// TIA Portal V16 export
// export: Created 2023-01-04T15:44:06.905709Z, ExportSetting WithDefaults, DisplayName Totally Integrated Automation Portal, DisplayVersion V16, DisplayName TIA Portal Version Control Interface, DisplayVersion V16, DisplayName TIA Portal Openness, DisplayVersion V16, DisplayName STEP 7 Professional, DisplayVersion V16, DisplayName STEP 7 Safety, DisplayVersion V16, DisplayName WinCC Advanced, DisplayVersion V16
FUNCTION "Filling_Logik" : Void   // FC5, LAD
{ S7_Optimized_Access := 'TRUE' }
VERSION : 0.1
// stored: AutoNumber true, IsIECCheckEnabled false, SetENOAutomatically false, UDAEnableTagReadback false
   VAR_INPUT
      PS2_Filling_Station : Bool;
      FIC_B102 : Int;
      Liquid_AorB_in_Bottle_ml : Real;
      Liquid_AorB_pct : Int;
      Wait_to_fill : Time;
   END_VAR
   VAR_OUTPUT
      Flow_ml_per_sec : Real;
      FillingData_LiqAorB_ml : Real;
   END_VAR
   VAR_IN_OUT
      Outlet_of_tanks : Bool;
   END_VAR
   VAR_TEMP
      PTRIG1 : Bool;
      PTRIG2 : Bool;
      PTRIG3 : Bool;
      PTRIG4 : Bool;
   END_VAR
BEGIN

REGION Network 1
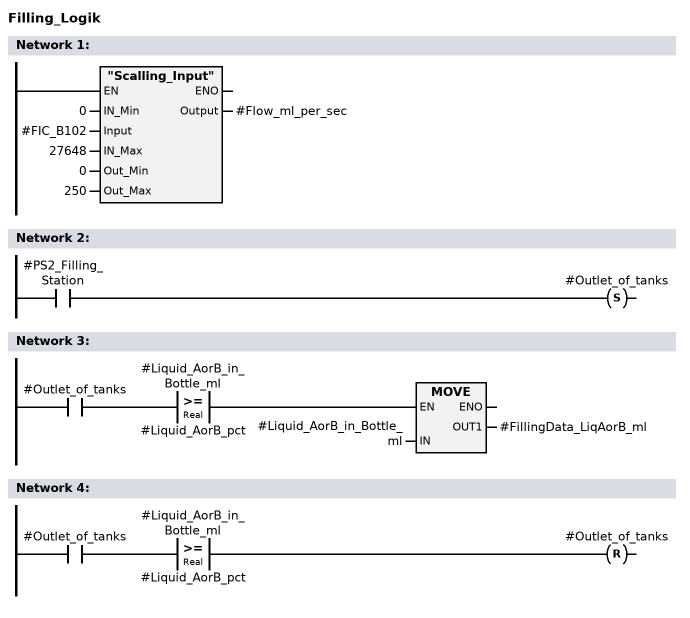
   RUNG wire#powerrail
      "Scalling_Input"(IN_Min := 0, Input := #FIC_B102, IN_Max := 27648, Out_Min := 0, Out_Max := 250, Output => #Flow_ml_per_sec)
   END_RUNG
   // the same network as SCL:
   "Scalling_Input"(IN_Min := 0,
                    Input := #FIC_B102,
                    IN_Max := 27648,
                    Out_Min := 0,
                    Out_Max := 250,
                    Output => #Flow_ml_per_sec);
END_REGION

REGION Network 2
   RUNG wire#powerrail
      Contact( #PS2_Filling_Station )
      S_Coil( #Outlet_of_tanks )
   END_RUNG
   // the same network as SCL:
   IF #PS2_Filling_Station THEN #Outlet_of_tanks := TRUE; END_IF;
END_REGION

REGION Network 3
   RUNG wire#powerrail
      Contact( #Outlet_of_tanks )
      { S7_Templates := "SrcType := Real" } GE_Contact(in1 := #Liquid_AorB_in_Bottle_ml, in2 := #Liquid_AorB_pct)
      Move(in := #Liquid_AorB_in_Bottle_ml, out1 => #FillingData_LiqAorB_ml)
   END_RUNG
   // the same network as SCL:
   IF #Outlet_of_tanks AND (#Liquid_AorB_in_Bottle_ml >= #Liquid_AorB_pct) THEN
       #FillingData_LiqAorB_ml := #Liquid_AorB_in_Bottle_ml;
   END_IF;
END_REGION

REGION Network 4
   RUNG wire#powerrail
      Contact( #Outlet_of_tanks )
      { S7_Templates := "SrcType := Real" } GE_Contact(in1 := #Liquid_AorB_in_Bottle_ml, in2 := #Liquid_AorB_pct)
      R_Coil( #Outlet_of_tanks )
   END_RUNG
   // the same network as SCL:
   IF #Outlet_of_tanks AND (#Liquid_AorB_in_Bottle_ml >= #Liquid_AorB_pct) THEN
       #Outlet_of_tanks := FALSE;
   END_IF;
END_REGION
END_FUNCTION
